// TIA Portal V17 export
// export: Created 2022-07-29T12:02:58.1165734Z, ExportSetting WithDefaults, DisplayName Totally Integrated Automation Portal, DisplayVersion V17 Update 4, DisplayName TIA Portal Openness, DisplayVersion V17 Update 4, DisplayName TIA Portal Teamcenter Gateway, DisplayVersion V17 Update 4, DisplayName TIA Portal Version Control Interface, DisplayVersion V17, DisplayName SINAMICS Startdrive Advanced, DisplayVersion V17 Update2, DisplayName SINAMICS Startdrive G130, G150, S120, S150, SINAMICS MV, S210, DisplayVersion V17 Update2, DisplayName SINAMICS Startdrive G110M, G120, G120C, G120D, G120P, G115D, DisplayVersion V17 Update2, DisplayName STEP 7 Professional, DisplayVersion V17 Update 4, DisplayName STEP 7 Safety, DisplayVersion V17, DisplayName WinCC Advanced / Unified PC, DisplayVersion V17 Update 4
ORGANIZATION_BLOCK "Main"   // OB1, LAD, ProgramCycle
TITLE = "Main Program Sweep (Cycle)"
{ S7_Optimized_Access := 'TRUE' }
VERSION : 0.1
// stored: AutoNumber true, IsIECCheckEnabled false, SetENOAutomatically false
   VAR_INPUT
      Initial_Call : Bool;   // Initial call of this OB
      Remanence : Bool;   // =True, if remanent data are available
   END_VAR
   VAR_TEMP
      temp_1 : Bool;
      temp_2 : Bool;
      "temp Int" : Int;
   END_VAR
   VAR_TEMP   // added for the SCL form of the ladder/FBD networks
      _w1 : Bool;
   END_VAR
BEGIN

REGION Network 1
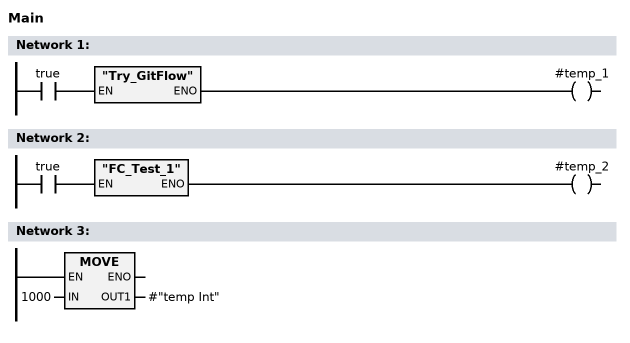
   RUNG wire#powerrail
      Contact( true )
      "Try_GitFlow"()
      Coil( #temp_1 )
   END_RUNG
   // the same network as SCL:
   "Try_GitFlow"(EN := true, ENO => #_w1);
   #temp_1 := #_w1;
END_REGION

REGION Network 2
   RUNG wire#powerrail
      Contact( true )
      "FC_Test_1"()
      Coil( #temp_2 )
   END_RUNG
   // the same network as SCL:
   "FC_Test_1"(EN := true, ENO => #_w1);
   #temp_2 := #_w1;
END_REGION

REGION Network 3
   RUNG wire#powerrail
      Move(in := 1000, out1 => #"temp Int")
   END_RUNG
   // the same network as SCL:
   #"temp Int" := 1000;
END_REGION
END_ORGANIZATION_BLOCK
